FUNCTION fDeg2Rad : REAL
VAR_INPUT
	fDeg : LREAL;
END_VAR
VAR
	
END_VAR

fDeg2Rad := fDeg * (3.14/180);

END_FUNCTION

(* stored: Version 1.1.0.1, ProductVersion 3.1.4024.12
   POU fDeg2Rad: Id {c367d73b-9ceb-4476-95a1-89bdb986e7cd}, SpecialFunc None *)
